(*
SPDX-FileCopyrightText: © 2026 Oleksandr Tiutyk <trofimich@gmail.com>
SPDX-License-Identifier: MIT
License: https://opensource.org/license/mit
*)

(*!
<summary>
Beckhoff EL6022: 2-channel serial interface terminal (RS422 / RS485).
</summary>
<description>
Process image mapping structure for the EL6022 2-channel serial interface terminal using 22-byte data
exchange.
When used for I/O, link located fields or their containing buffers to the matching selected PDOs.
The record is not a packed wire buffer; compiler padding is not part of the device specification.
Unlinked/default values do not prove valid I/O. The caller evaluates bus/channel validity before use.
Use one owner task per instance and externally synchronize other access; multi-field snapshots are not atomic.
Copies store data without creating hardware links. Keep borrowed field references valid while consumers are bound.
This passive record performs no validation, synchronization, configuration or protocol advancement.
Select the 22-byte serial payload with 16-bit status/control words; larger buffers and 9-bit modes
are outside this model. The owning service implements the transmit/receive toggle handshake.
</description>
*)
TYPE EL6022 :
STRUCT
	Ch1 : EL6022_CHANNEL;
	Ch2 : EL6022_CHANNEL;
END_STRUCT
END_TYPE

(* stored: Version 1.1.0.1, ProductVersion 3.1.4026.20
   DUT EL6022: Id {3bfb6762-705e-45d9-b3d0-da51074e3bf1} *)
